FUNCTION StopPump : BOOL
VAR_IN_OUT
	Pump		:	PumpType;
END_VAR
VAR
END_VAR

// pump will stop after 30 sec delay to avoid unnecessary start/stop

IF Pump.RunLastStartSec > 5 THEN
	Pump.RunState := PumpState.STOP;
	Pump.RunLastStartSec := 0;
END_IF

END_FUNCTION

(* stored: Version 1.1.0.1, ProductVersion 3.1.4024.15
   POU StopPump: Id {9bd54186-fdba-49c2-b637-117b8f41f4cd}, SpecialFunc None *)
